// TIA Portal V19 export
FUNCTION_BLOCK "Valve"   // FB120, LAD
TITLE = VALVE MANAGER / Valve Management FB
AUTHOR : PIH
FAMILY : Devices
VERSION : 1.94
// stored: Access Published, MemoryReserve 100, SetENOAutomatically false
   VAR_INPUT
      ValveCtrl : "ValveCtrl";
      RestLimitSwitch : Bool;   // Rest limit switch
      WorkLimitSwitch : Bool;   // Work limit switch
      OilInPressure : Bool;   // Oil in pressure (only for oil valve)
      Simulation : Bool;
      Config : "ValveConfig";   // configurations & parameters
   END_VAR
   VAR_OUTPUT
      ValveSts : "ValveSts";
      RestSolenoid : Bool;
      WorkSolenoid : Bool;
      ReqOilPressure : Bool;   // Request oli pressure to Hydraulic unit (only for oil valve)
   END_VAR
   VAR_IN_OUT
      Alarm : "ValveAlr";
   END_VAR
   VAR DB_SPECIFIC
      IsAtRest : Bool;
      IsAtWork : Bool;
   END_VAR
   VAR
      Ctrl : Struct
         RestReq : Bool;
         WorkReq : Bool;
         RestSolenoid : Bool;
         WorkSolenoid : Bool;
      END_STRUCT;
      tonRest : IEC_TIMER;
      tonWork : IEC_TIMER;
      tonTimeOutRest : IEC_TIMER;
      tonTimeOutWork : IEC_TIMER;
   END_VAR
   VAR_TEMP
      RestAlarmsPresence : Bool;
      RestPermitted : Bool;
      WorkAlarmsPresence : Bool;
      WorkPermitted : Bool;
      CheckTOutRest : Bool;
      CheckTOutWork : Bool;
   END_VAR
BEGIN

REGION Network 1 (SCL): Info
   //=============================================================================
   //PM FORMING
   //-----------------------------------------------------------------------------
   // Library: StandardBlocks
   // Tested with: S7-1518TF
   // Engineering: TIA Portal V18
   // Restrictions: -
   // Requirements: S7-1500
   // Functionality: Valve device manager
   //
   // v1.0.0  28/12/2022 
   // v1.1.0  23/01/2023 Simulation added
   // v1.1.1  14/02/2022 Config udt added
   //=============================================================================
END_REGION

REGION Network 2: Time for valve at rest status
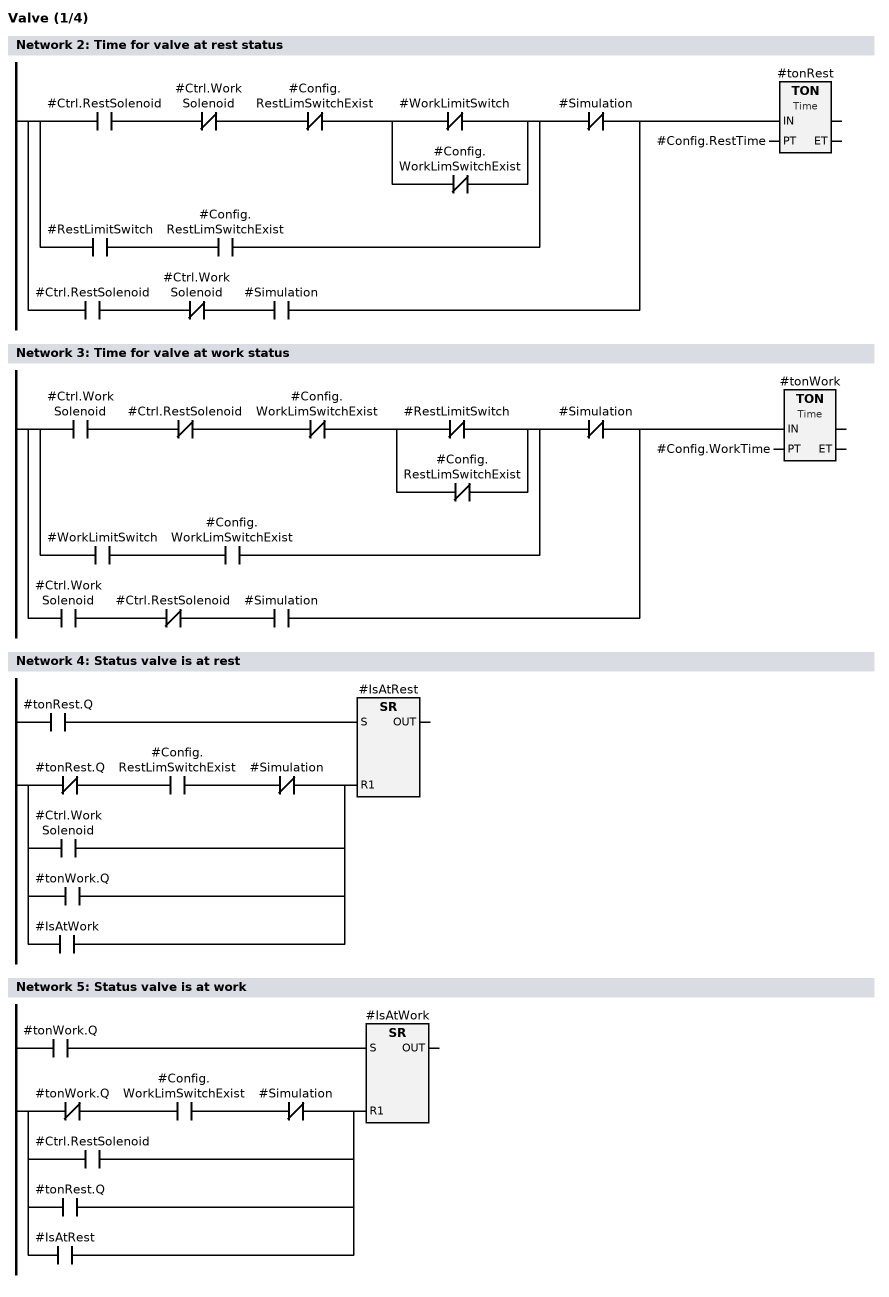
   RUNG wire#powerrail
      Contact( #Ctrl.RestSolenoid )
      I_Contact( #Ctrl.WorkSolenoid )
      I_Contact( #Config.RestLimSwitchExist )
      wire#w1
      I_Contact( #WorkLimitSwitch )
      wire#w2
      I_Contact( #Simulation )
      wire#w3
      { S7_Templates := "time_type := Time" } #tonRest.TON(pt := #Config.RestTime, et =>)
   END_RUNG
   RUNG wire#w1
      I_Contact( #Config.WorkLimSwitchExist )
   END_RUNG wire#w2
   RUNG wire#powerrail
      Contact( #RestLimitSwitch )
      Contact( #Config.RestLimSwitchExist )
   END_RUNG wire#w2
   RUNG wire#powerrail
      Contact( #Ctrl.RestSolenoid )
      I_Contact( #Ctrl.WorkSolenoid )
      Contact( #Simulation )
   END_RUNG wire#w3
   // the same network as SCL:
   #tonRest.TON(IN := (((#Ctrl.RestSolenoid AND NOT #Ctrl.WorkSolenoid AND NOT #Config.RestLimSwitchExist AND (NOT #WorkLimitSwitch OR NOT #Config.WorkLimSwitchExist)) OR (#RestLimitSwitch AND #Config.RestLimSwitchExist)) AND NOT #Simulation) OR (#Ctrl.RestSolenoid AND NOT #Ctrl.WorkSolenoid AND #Simulation),
                PT := #Config.RestTime);
END_REGION

REGION Network 3: Time for valve at work status
   RUNG wire#powerrail
      Contact( #Ctrl.WorkSolenoid )
      I_Contact( #Ctrl.RestSolenoid )
      I_Contact( #Config.WorkLimSwitchExist )
      wire#w1
      I_Contact( #RestLimitSwitch )
      wire#w2
      I_Contact( #Simulation )
      wire#w3
      { S7_Templates := "time_type := Time" } #tonWork.TON(pt := #Config.WorkTime, et =>)
   END_RUNG
   RUNG wire#w1
      I_Contact( #Config.RestLimSwitchExist )
   END_RUNG wire#w2
   RUNG wire#powerrail
      Contact( #WorkLimitSwitch )
      Contact( #Config.WorkLimSwitchExist )
   END_RUNG wire#w2
   RUNG wire#powerrail
      Contact( #Ctrl.WorkSolenoid )
      I_Contact( #Ctrl.RestSolenoid )
      Contact( #Simulation )
   END_RUNG wire#w3
   // the same network as SCL:
   #tonWork.TON(IN := (((#Ctrl.WorkSolenoid AND NOT #Ctrl.RestSolenoid AND NOT #Config.WorkLimSwitchExist AND (NOT #RestLimitSwitch OR NOT #Config.RestLimSwitchExist)) OR (#WorkLimitSwitch AND #Config.WorkLimSwitchExist)) AND NOT #Simulation) OR (#Ctrl.WorkSolenoid AND NOT #Ctrl.RestSolenoid AND #Simulation),
                PT := #Config.WorkTime);
END_REGION

REGION Network 4: Status valve is at rest
   RUNG wire#powerrail
      Contact( #tonRest.Q )
      S_SR(operand := #IsAtRest, r1 := wire#w1)
   END_RUNG
   RUNG wire#powerrail
      I_Contact( #tonRest.Q )
      Contact( #Config.RestLimSwitchExist )
      I_Contact( #Simulation )
   END_RUNG wire#w1
   RUNG wire#powerrail
      Contact( #Ctrl.WorkSolenoid )
   END_RUNG wire#w1
   RUNG wire#powerrail
      Contact( #tonWork.Q )
   END_RUNG wire#w1
   RUNG wire#powerrail
      Contact( #IsAtWork )
   END_RUNG wire#w1
   // the same network as SCL:
   IF #tonRest.Q THEN
       #IsAtRest := TRUE;   // SR flip-flop
   END_IF;
   IF (NOT #tonRest.Q AND #Config.RestLimSwitchExist AND NOT #Simulation) OR #Ctrl.WorkSolenoid OR #tonWork.Q OR #IsAtWork THEN
       #IsAtRest := FALSE;
   END_IF;
END_REGION

REGION Network 5: Status valve is at work
   RUNG wire#powerrail
      Contact( #tonWork.Q )
      S_SR(operand := #IsAtWork, r1 := wire#w1)
   END_RUNG
   RUNG wire#powerrail
      I_Contact( #tonWork.Q )
      Contact( #Config.WorkLimSwitchExist )
      I_Contact( #Simulation )
   END_RUNG wire#w1
   RUNG wire#powerrail
      Contact( #Ctrl.RestSolenoid )
   END_RUNG wire#w1
   RUNG wire#powerrail
      Contact( #tonRest.Q )
   END_RUNG wire#w1
   RUNG wire#powerrail
      Contact( #IsAtRest )
   END_RUNG wire#w1
   // the same network as SCL:
   IF #tonWork.Q THEN
       #IsAtWork := TRUE;   // SR flip-flop
   END_IF;
   IF (NOT #tonWork.Q AND #Config.WorkLimSwitchExist AND NOT #Simulation) OR #Ctrl.RestSolenoid OR #tonRest.Q OR #IsAtRest THEN
       #IsAtWork := FALSE;
   END_IF;
END_REGION

REGION Network 6: <<< ALARMS >>>
END_REGION

REGION Network 7: Time for check timeout rest / Time for check timeout
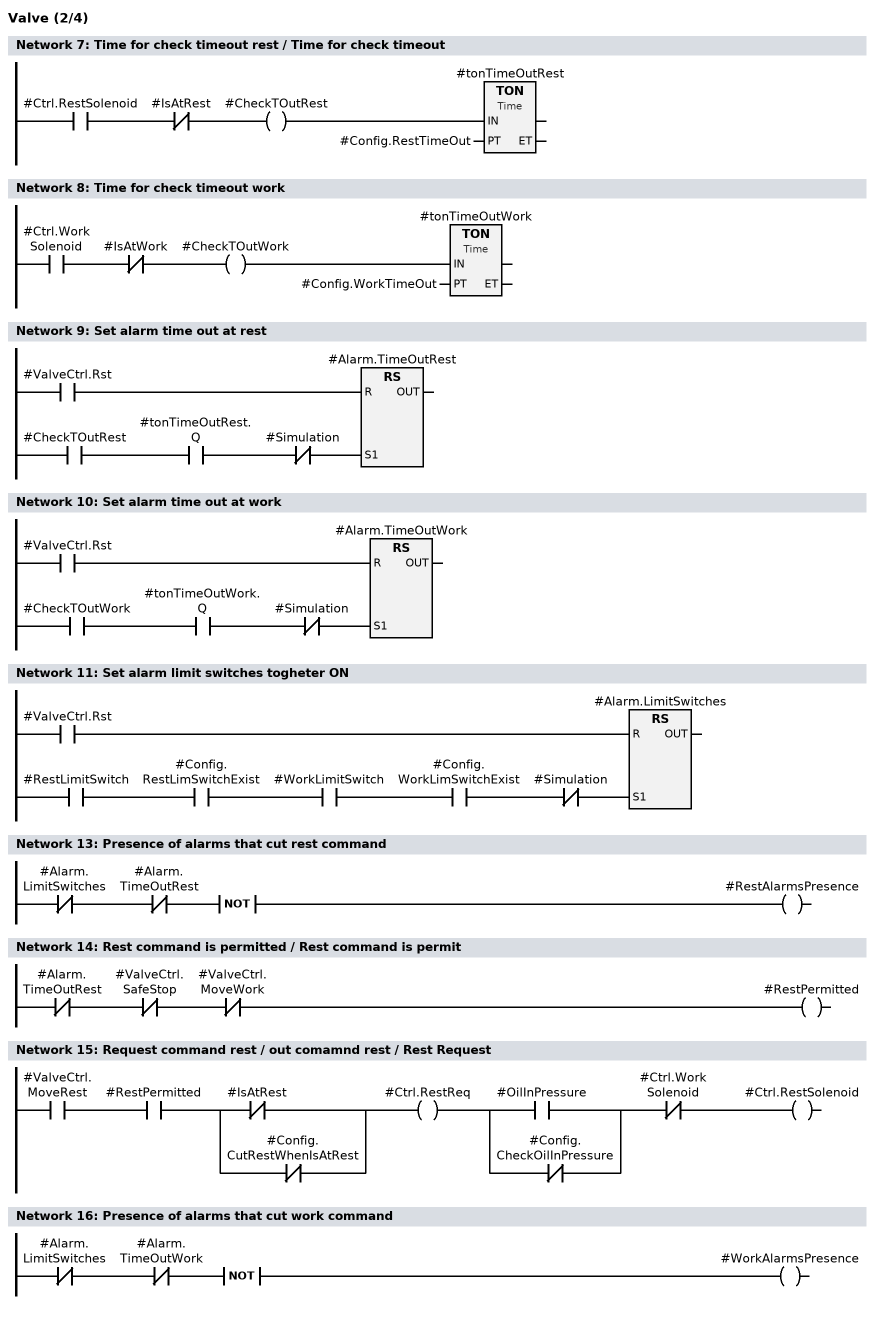
   RUNG wire#powerrail
      Contact( #Ctrl.RestSolenoid )
      I_Contact( #IsAtRest )
      Coil( #CheckTOutRest )
      { S7_Templates := "time_type := Time" } #tonTimeOutRest.TON(pt := #Config.RestTimeOut, et =>)
   END_RUNG
   // the same network as SCL:
   #CheckTOutRest := #Ctrl.RestSolenoid AND NOT #IsAtRest;
   #tonTimeOutRest.TON(IN := #CheckTOutRest, PT := #Config.RestTimeOut);
END_REGION

REGION Network 8: Time for check timeout work
   RUNG wire#powerrail
      Contact( #Ctrl.WorkSolenoid )
      I_Contact( #IsAtWork )
      Coil( #CheckTOutWork )
      { S7_Templates := "time_type := Time" } #tonTimeOutWork.TON(pt := #Config.WorkTimeOut, et =>)
   END_RUNG
   // the same network as SCL:
   #CheckTOutWork := #Ctrl.WorkSolenoid AND NOT #IsAtWork;
   #tonTimeOutWork.TON(IN := #CheckTOutWork, PT := #Config.WorkTimeOut);
END_REGION

REGION Network 9: Set alarm time out at rest
   RUNG wire#powerrail
      Contact( #ValveCtrl.Rst )
      S_RS(operand := #Alarm.TimeOutRest, s1 := wire#w1)
   END_RUNG
   RUNG wire#powerrail
      Contact( #CheckTOutRest )
      Contact( #tonTimeOutRest.Q )
      I_Contact( #Simulation )
   END_RUNG wire#w1
   // the same network as SCL:
   IF #ValveCtrl.Rst THEN
       #Alarm.TimeOutRest := FALSE;   // RS flip-flop
   END_IF;
   IF #CheckTOutRest AND #tonTimeOutRest.Q AND NOT #Simulation THEN #Alarm.TimeOutRest := TRUE; END_IF;
END_REGION

REGION Network 10: Set alarm time out at work
   RUNG wire#powerrail
      Contact( #ValveCtrl.Rst )
      S_RS(operand := #Alarm.TimeOutWork, s1 := wire#w1)
   END_RUNG
   RUNG wire#powerrail
      Contact( #CheckTOutWork )
      Contact( #tonTimeOutWork.Q )
      I_Contact( #Simulation )
   END_RUNG wire#w1
   // the same network as SCL:
   IF #ValveCtrl.Rst THEN
       #Alarm.TimeOutWork := FALSE;   // RS flip-flop
   END_IF;
   IF #CheckTOutWork AND #tonTimeOutWork.Q AND NOT #Simulation THEN #Alarm.TimeOutWork := TRUE; END_IF;
END_REGION

REGION Network 11: Set alarm limit switches togheter ON
   RUNG wire#powerrail
      Contact( #ValveCtrl.Rst )
      S_RS(operand := #Alarm.LimitSwitches, s1 := wire#w1)
   END_RUNG
   RUNG wire#powerrail
      Contact( #RestLimitSwitch )
      Contact( #Config.RestLimSwitchExist )
      Contact( #WorkLimitSwitch )
      Contact( #Config.WorkLimSwitchExist )
      I_Contact( #Simulation )
   END_RUNG wire#w1
   // the same network as SCL:
   IF #ValveCtrl.Rst THEN
       #Alarm.LimitSwitches := FALSE;   // RS flip-flop
   END_IF;
   IF #RestLimitSwitch AND #Config.RestLimSwitchExist AND #WorkLimitSwitch AND #Config.WorkLimSwitchExist AND NOT #Simulation THEN
       #Alarm.LimitSwitches := TRUE;
   END_IF;
END_REGION

REGION Network 12: <<< COMMANDS >>>
END_REGION

REGION Network 13: Presence of alarms that cut rest command
   RUNG wire#powerrail
      I_Contact( #Alarm.LimitSwitches )
      I_Contact( #Alarm.TimeOutRest )
      Not()
      Coil( #RestAlarmsPresence )
   END_RUNG
   // the same network as SCL:
   #RestAlarmsPresence := NOT (NOT #Alarm.LimitSwitches AND NOT #Alarm.TimeOutRest);
END_REGION

REGION Network 14: Rest command is permitted / Rest command is permit
   RUNG wire#powerrail
      I_Contact( #Alarm.TimeOutRest )
      I_Contact( #ValveCtrl.SafeStop )
      I_Contact( #ValveCtrl.MoveWork )
      Coil( #RestPermitted )
   END_RUNG
   // the same network as SCL:
   #RestPermitted := NOT #Alarm.TimeOutRest AND NOT #ValveCtrl.SafeStop AND NOT #ValveCtrl.MoveWork;
END_REGION

REGION Network 15: Request command rest / out comamnd rest / Rest Request
   RUNG wire#powerrail
      Contact( #ValveCtrl.MoveRest )
      Contact( #RestPermitted )
      wire#w1
      I_Contact( #IsAtRest )
      wire#w2
      Coil( #Ctrl.RestReq )
      wire#w3
      Contact( #OilInPressure )
      wire#w4
      I_Contact( #Ctrl.WorkSolenoid )
      Coil( #Ctrl.RestSolenoid )
   END_RUNG
   RUNG wire#w1
      I_Contact( #Config.CutRestWhenIsAtRest )
   END_RUNG wire#w2
   RUNG wire#w3
      I_Contact( #Config.CheckOilInPressure )
   END_RUNG wire#w4
   // the same network as SCL:
   #Ctrl.RestReq := #ValveCtrl.MoveRest AND #RestPermitted AND (NOT #IsAtRest OR NOT #Config.CutRestWhenIsAtRest);
   #Ctrl.RestSolenoid := #Ctrl.RestReq AND (#OilInPressure OR NOT #Config.CheckOilInPressure) AND NOT #Ctrl.WorkSolenoid;
END_REGION

REGION Network 16: Presence of alarms that cut work command
   RUNG wire#powerrail
      I_Contact( #Alarm.LimitSwitches )
      I_Contact( #Alarm.TimeOutWork )
      Not()
      Coil( #WorkAlarmsPresence )
   END_RUNG
   // the same network as SCL:
   #WorkAlarmsPresence := NOT (NOT #Alarm.LimitSwitches AND NOT #Alarm.TimeOutWork);
END_REGION

REGION Network 17: Work command is permitted / Work command is permit
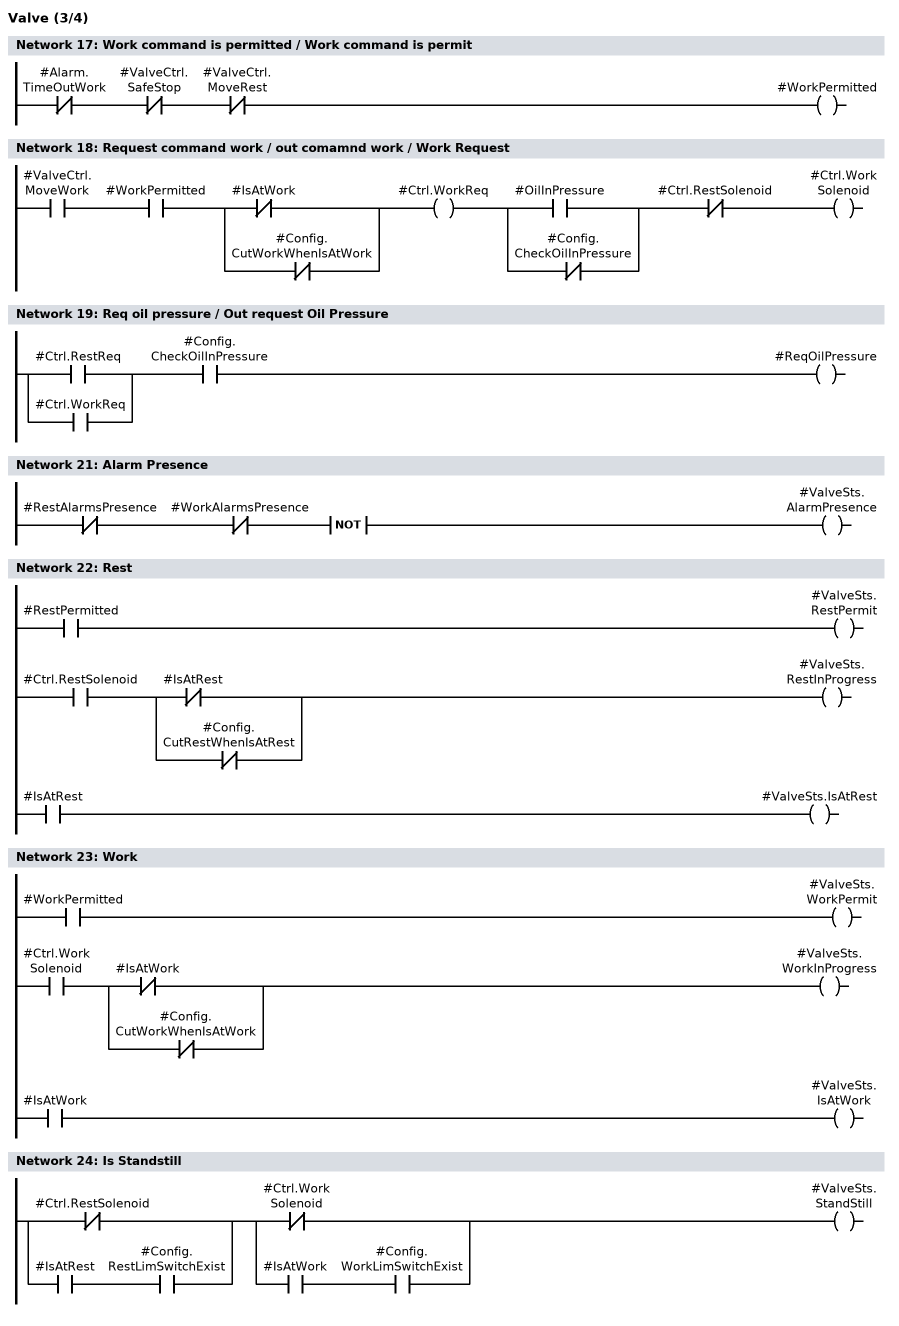
   RUNG wire#powerrail
      I_Contact( #Alarm.TimeOutWork )
      I_Contact( #ValveCtrl.SafeStop )
      I_Contact( #ValveCtrl.MoveRest )
      Coil( #WorkPermitted )
   END_RUNG
   // the same network as SCL:
   #WorkPermitted := NOT #Alarm.TimeOutWork AND NOT #ValveCtrl.SafeStop AND NOT #ValveCtrl.MoveRest;
END_REGION

REGION Network 18: Request command work / out comamnd work / Work Request
   RUNG wire#powerrail
      Contact( #ValveCtrl.MoveWork )
      Contact( #WorkPermitted )
      wire#w1
      I_Contact( #IsAtWork )
      wire#w2
      Coil( #Ctrl.WorkReq )
      wire#w3
      Contact( #OilInPressure )
      wire#w4
      I_Contact( #Ctrl.RestSolenoid )
      Coil( #Ctrl.WorkSolenoid )
   END_RUNG
   RUNG wire#w1
      I_Contact( #Config.CutWorkWhenIsAtWork )
   END_RUNG wire#w2
   RUNG wire#w3
      I_Contact( #Config.CheckOilInPressure )
   END_RUNG wire#w4
   // the same network as SCL:
   #Ctrl.WorkReq := #ValveCtrl.MoveWork AND #WorkPermitted AND (NOT #IsAtWork OR NOT #Config.CutWorkWhenIsAtWork);
   #Ctrl.WorkSolenoid := #Ctrl.WorkReq AND (#OilInPressure OR NOT #Config.CheckOilInPressure) AND NOT #Ctrl.RestSolenoid;
END_REGION

REGION Network 19: Req oil pressure / Out request Oil Pressure
   RUNG wire#powerrail
      Contact( #Ctrl.RestReq )
      wire#w1
      Contact( #Config.CheckOilInPressure )
      Coil( #ReqOilPressure )
   END_RUNG
   RUNG wire#powerrail
      Contact( #Ctrl.WorkReq )
   END_RUNG wire#w1
   // the same network as SCL:
   #ReqOilPressure := (#Ctrl.RestReq OR #Ctrl.WorkReq) AND #Config.CheckOilInPressure;
END_REGION

REGION Network 20: <<< STATUS >>>
END_REGION

REGION Network 21: Alarm Presence
   RUNG wire#powerrail
      I_Contact( #RestAlarmsPresence )
      I_Contact( #WorkAlarmsPresence )
      Not()
      Coil( #ValveSts.AlarmPresence )
   END_RUNG
   // the same network as SCL:
   #ValveSts.AlarmPresence := NOT (NOT #RestAlarmsPresence AND NOT #WorkAlarmsPresence);
END_REGION

REGION Network 22: Rest
   RUNG wire#powerrail
      Contact( #RestPermitted )
      Coil( #ValveSts.RestPermit )
   END_RUNG
   RUNG wire#powerrail
      Contact( #Ctrl.RestSolenoid )
      wire#w1
      I_Contact( #IsAtRest )
      wire#w2
      Coil( #ValveSts.RestInProgress )
   END_RUNG
   RUNG wire#w1
      I_Contact( #Config.CutRestWhenIsAtRest )
   END_RUNG wire#w2
   RUNG wire#powerrail
      Contact( #IsAtRest )
      Coil( #ValveSts.IsAtRest )
   END_RUNG
   // the same network as SCL:
   #ValveSts.RestPermit := #RestPermitted;
   #ValveSts.RestInProgress := #Ctrl.RestSolenoid AND (NOT #IsAtRest OR NOT #Config.CutRestWhenIsAtRest);
   #ValveSts.IsAtRest := #IsAtRest;
END_REGION

REGION Network 23: Work
   RUNG wire#powerrail
      Contact( #WorkPermitted )
      Coil( #ValveSts.WorkPermit )
   END_RUNG
   RUNG wire#powerrail
      Contact( #Ctrl.WorkSolenoid )
      wire#w1
      I_Contact( #IsAtWork )
      wire#w2
      Coil( #ValveSts.WorkInProgress )
   END_RUNG
   RUNG wire#w1
      I_Contact( #Config.CutWorkWhenIsAtWork )
   END_RUNG wire#w2
   RUNG wire#powerrail
      Contact( #IsAtWork )
      Coil( #ValveSts.IsAtWork )
   END_RUNG
   // the same network as SCL:
   #ValveSts.WorkPermit := #WorkPermitted;
   #ValveSts.WorkInProgress := #Ctrl.WorkSolenoid AND (NOT #IsAtWork OR NOT #Config.CutWorkWhenIsAtWork);
   #ValveSts.IsAtWork := #IsAtWork;
END_REGION

REGION Network 24: Is Standstill
   RUNG wire#powerrail
      I_Contact( #Ctrl.RestSolenoid )
      wire#w1
      I_Contact( #Ctrl.WorkSolenoid )
      wire#w2
      Coil( #ValveSts.StandStill )
   END_RUNG
   RUNG wire#powerrail
      Contact( #IsAtRest )
      Contact( #Config.RestLimSwitchExist )
   END_RUNG wire#w1
   RUNG wire#w1
      Contact( #IsAtWork )
      Contact( #Config.WorkLimSwitchExist )
   END_RUNG wire#w2
   // the same network as SCL:
   #ValveSts.StandStill := (NOT #Ctrl.RestSolenoid OR (#IsAtRest AND #Config.RestLimSwitchExist)) AND (NOT #Ctrl.WorkSolenoid OR (#IsAtWork AND #Config.WorkLimSwitchExist));
END_REGION

REGION Network 25: Out
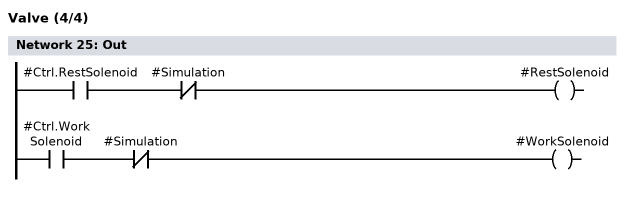
   RUNG wire#powerrail
      Contact( #Ctrl.RestSolenoid )
      I_Contact( #Simulation )
      Coil( #RestSolenoid )
   END_RUNG
   RUNG wire#powerrail
      Contact( #Ctrl.WorkSolenoid )
      I_Contact( #Simulation )
      Coil( #WorkSolenoid )
   END_RUNG
   // the same network as SCL:
   #RestSolenoid := #Ctrl.RestSolenoid AND NOT #Simulation;
   #WorkSolenoid := #Ctrl.WorkSolenoid AND NOT #Simulation;
END_REGION
END_FUNCTION_BLOCK
